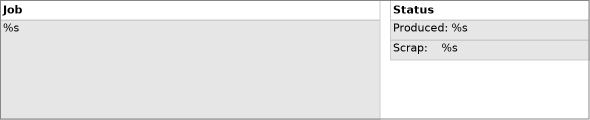
VISUALIZATION _VISU_ProductionOverview  // 590x120
VAR_IN_OUT
	mInst : FB_ProdManager_DMAX;
END_VAR
    Rectangle (0,20 380x100), "%s", text variable: mInst.sActiveJobInfo, colour toggle: mInst.bPmActive
    RoundedRectangle (0,0 380x20), "Job"
    RoundedRectangle (390,0 200x20), "Status"
    Rectangle (390,20 200x20), "Produced: %s", text variable: mInst.nProduced, colour toggle: mInst.nProduced > 0
    Rectangle (390,40 200x20), "Scrap: %s", text variable: mInst.nScrap, colour toggle: mInst.nScrap > 0
END_VISUALIZATION

(* stored: Version 1.1.0.1, ProductVersion 3.1.4024.11
   Visu _VISU_ProductionOverview: Id {d55e14b7-2896-443e-9edd-692d55843043} *)
